(* Logix 5000 project; controller ACIM5010ConveyorHailee_Renkers vendor 1 type 14 code 77 rev 20.12; software revision 20.01 *)

TASK MainTask (continuous, watchdog 500 ms) : MainProgram

MODULES
   Controller : vendor 1 type 14 code 77 (CompactLogixL32EController 0, rev 20.12)
      LocalENB : 1769-L32E Ethernet Port (CompactLogixL32Ethernet 1, rev 20.11)
      Local : CompactBus (CompactVirtualAdapter 3, rev 20.11)
         Inputmod : 1769-IQ16 (Compact 1, rev 1.1, Input RPI 20 ms)
         OutputMod : 1769-OW16 (Compact 2, rev 1.1, Output RPI 20 ms)
END_MODULES

VAR_GLOBAL   (* controller tags *)
   Bin_Left_Red_Light : ALIAS FOR Local:2:O.Data.3;
   Bin_Right_Red_Light : ALIAS FOR Local:2:O.Data.4;
   CONVEYOR_AUX : ALIAS FOR Local:1:I.Data.12;
   CONVEYOR_MOTOR : ALIAS FOR Local:2:O.Data.2;
   FORWARD_AUX : ALIAS FOR Local:1:I.Data.10;
   FORWARD_MOTOR : ALIAS FOR Local:2:O.Data.0;
   GREEN_LIGHT : ALIAS FOR Local:2:O.Data.6;
   Limit_Switch_Left : ALIAS FOR Local:1:I.Data.13;
   Limit_Switch_Right : ALIAS FOR Local:1:I.Data.14;
   PHOTOEYE : ALIAS FOR Local:1:I.Data.15;
   REVERSE_AUX : ALIAS FOR Local:1:I.Data.11;
   REVERSE_MOTOR : ALIAS FOR Local:2:O.Data.1;
   START_PB : ALIAS FOR Local:1:I.Data.9;
   STOP_PB : ALIAS FOR Local:1:I.Data.8;
   YELLOW_LIGHT : ALIAS FOR Local:2:O.Data.5;
END_VAR

PROGRAM MainProgram   (* main routine MainRoutine *)
VAR
   counter : COUNTER := (PRE := 4);
   done : COUNTER := (PRE := 4);
   Latch : BOOL;
   Latch2 : BOOL;
   left : BOOL;
   left_bit_check : BOOL;
   left_latch : BOOL;
   lls_i : BOOL;
   OFF_DELAY : TIMER := (PRE := 1000);
   ON_DELAY : TIMER := (PRE := 1000);
   ONESHOTTIMER : BOOL;
   PI_Counter : COUNTER := (PRE := 8);
   pie_i : BOOL;
   PROCESS_COUNTER : COUNTER := (PRE := 4);
   right : BOOL;
   right_bit_check : BOOL;
   right_latch : BOOL;
   rls_i : BOOL;
   S0 : BOOL;
   S0_x : BOOL;
   S1 : BOOL;
   S1_x : BOOL;
   S2 : BOOL;
   S2_x : BOOL;
   S3 : BOOL;
   S3_x : BOOL;
   S4 : BOOL;
   S4_x : BOOL;
   S5 : BOOL;
   S5_x : BOOL;
   S6 : BOOL;
   S6_x : BOOL;
   start_i : BOOL;
   stop_i : BOOL;
END_VAR

ROUTINE MainRoutine   (* ladder *)
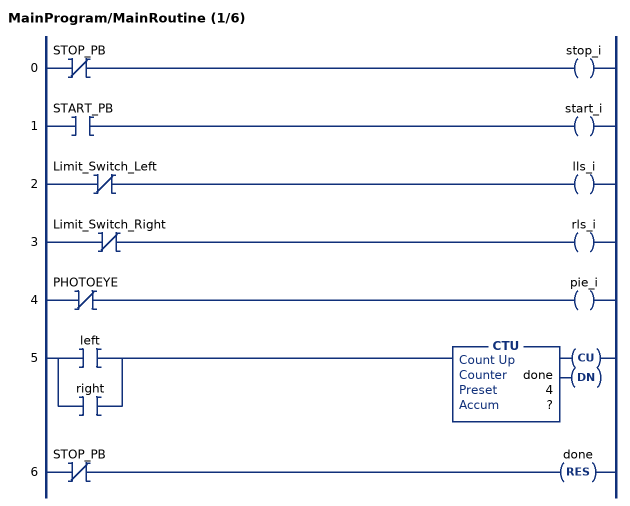
   0: XIO(STOP_PB)OTE(stop_i);
   1: XIC(START_PB)OTE(start_i);
   2: XIO(Limit_Switch_Left)OTE(lls_i);
   3: XIO(Limit_Switch_Right)OTE(rls_i);
   4: XIO(PHOTOEYE)OTE(pie_i);
   5: [XIC(left) ,XIC(right) ]CTU(done,?,?);
   6: XIO(STOP_PB)RES(done);
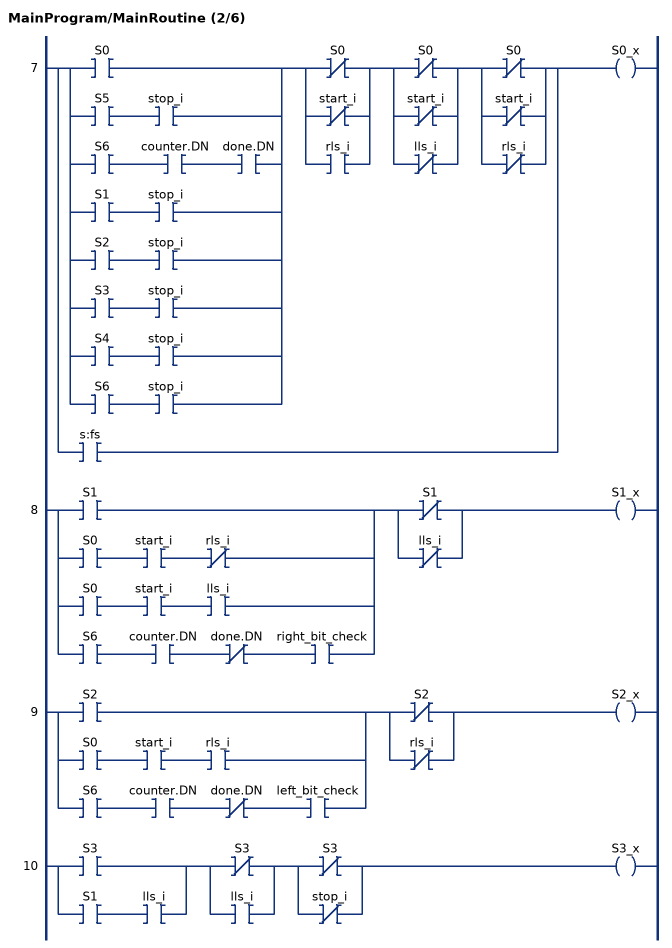
   7: [[XIC(S0) ,XIC(S5) XIC(stop_i) ,XIC(S6) XIC(counter.DN) XIC(done.DN) ,XIC(S1) XIC(stop_i) ,XIC(S2) XIC(stop_i) ,XIC(S3) XIC(stop_i) ,XIC(S4) XIC(stop_i) ,XIC(S6) XIC(stop_i) ] [XIO(S0) ,XIO(start_i) ,XIC(rls_i) ] [XIO(S0) ,XIO(start_i) ,XIO(lls_i) ] [XIO(S0) ,XIO(start_i) ,XIO(rls_i) ] ,XIC(s:fs) ]OTE(S0_x);
   8: [XIC(S1) ,[XIC(S0) XIC(start_i) XIO(rls_i) ,XIC(S0) XIC(start_i) XIC(lls_i) ] ,XIC(S6) XIC(counter.DN) XIO(done.DN) XIC(right_bit_check) ][XIO(S1) ,XIO(lls_i) ]OTE(S1_x);
   9: [XIC(S2) ,XIC(S0) XIC(start_i) XIC(rls_i) ,XIC(S6) XIC(counter.DN) XIO(done.DN) XIC(left_bit_check) ][XIO(S2) ,XIO(rls_i) ]OTE(S2_x);
   10: [XIC(S3) ,XIC(S1) XIC(lls_i) ][XIO(S3) ,XIC(lls_i) ][XIO(S3) ,XIO(stop_i) ]OTE(S3_x);
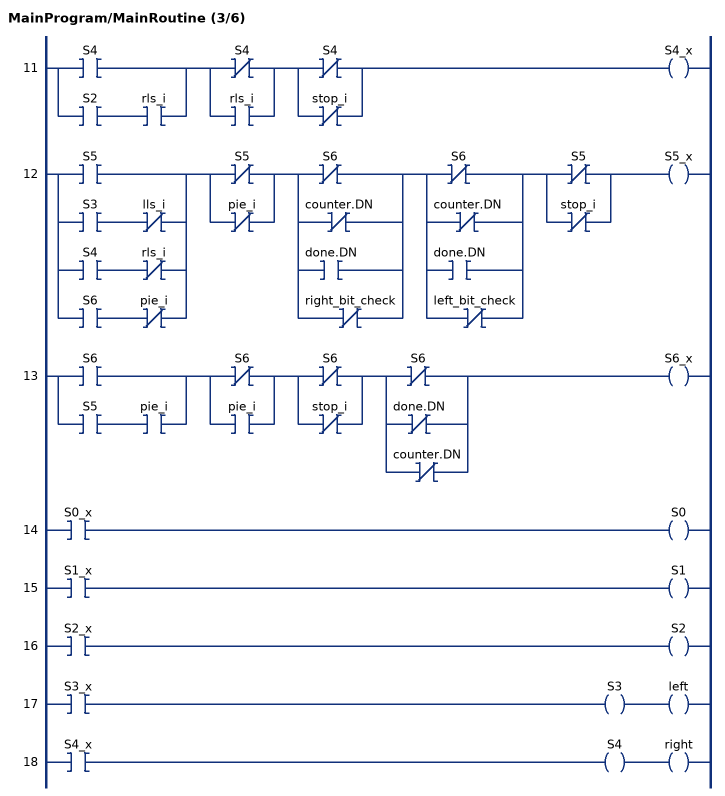
   11: [XIC(S4) ,XIC(S2) XIC(rls_i) ][XIO(S4) ,XIC(rls_i) ][XIO(S4) ,XIO(stop_i) ]OTE(S4_x);
   12: [XIC(S5) ,XIC(S3) XIO(lls_i) ,XIC(S4) XIO(rls_i) ,XIC(S6) XIO(pie_i) ][XIO(S5) ,XIO(pie_i) ][XIO(S6) ,XIO(counter.DN) ,XIC(done.DN) ,XIO(right_bit_check) ][XIO(S6) ,XIO(counter.DN) ,XIC(done.DN) ,XIO(left_bit_check) ][XIO(S5) ,XIO(stop_i) ]OTE(S5_x);
   13: [XIC(S6) ,XIC(S5) XIC(pie_i) ][XIO(S6) ,XIC(pie_i) ][XIO(S6) ,XIO(stop_i) ][XIO(S6) ,XIO(done.DN) ,XIO(counter.DN) ]OTE(S6_x);
   14: XIC(S0_x)OTE(S0);
   15: XIC(S1_x)OTE(S1);
   16: XIC(S2_x)OTE(S2);
   17: XIC(S3_x)OTE(S3)OTE(left);
   18: XIC(S4_x)OTE(S4)OTE(right);
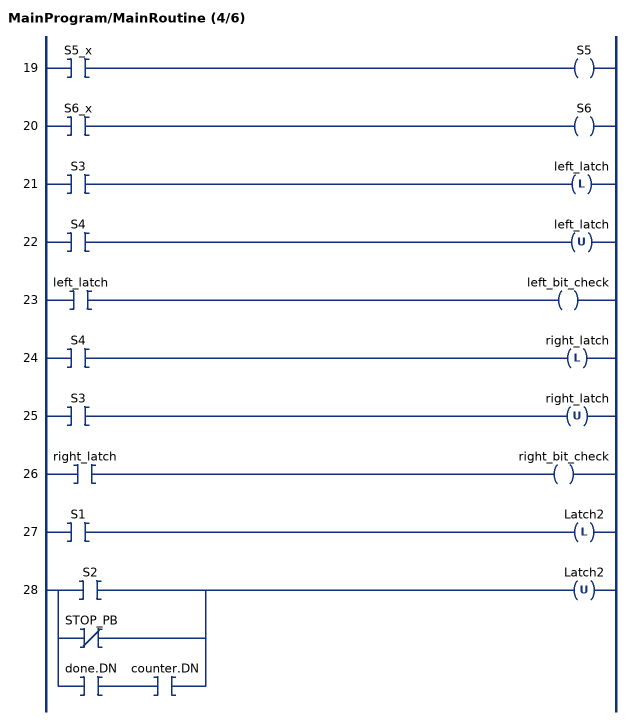
   19: XIC(S5_x)OTE(S5);
   20: XIC(S6_x)OTE(S6);
   21: XIC(S3)OTL(left_latch);
   22: XIC(S4)OTU(left_latch);
   23: XIC(left_latch)OTE(left_bit_check);
   24: XIC(S4)OTL(right_latch);
   25: XIC(S3)OTU(right_latch);
   26: XIC(right_latch)OTE(right_bit_check);
   27: XIC(S1)OTL(Latch2);
   28: [XIC(S2) ,XIO(STOP_PB) ,XIC(done.DN) XIC(counter.DN) ]OTU(Latch2);
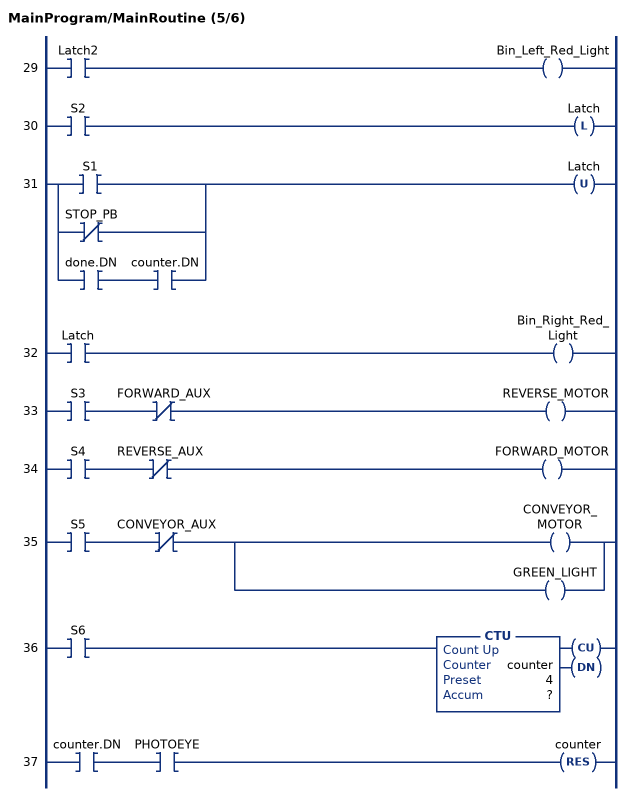
   29: XIC(Latch2)OTE(Bin_Left_Red_Light);
   30: XIC(S2)OTL(Latch);
   31: [XIC(S1) ,XIO(STOP_PB) ,XIC(done.DN) XIC(counter.DN) ]OTU(Latch);
   32: XIC(Latch)OTE(Bin_Right_Red_Light);
   33: XIC(S3)XIO(FORWARD_AUX)OTE(REVERSE_MOTOR);
   34: XIC(S4)XIO(REVERSE_AUX)OTE(FORWARD_MOTOR);
   35: XIC(S5)XIO(CONVEYOR_AUX)[OTE(CONVEYOR_MOTOR) ,OTE(GREEN_LIGHT) ];
   36: XIC(S6)CTU(counter,?,?);
   37: XIC(counter.DN)XIC(PHOTOEYE)RES(counter);
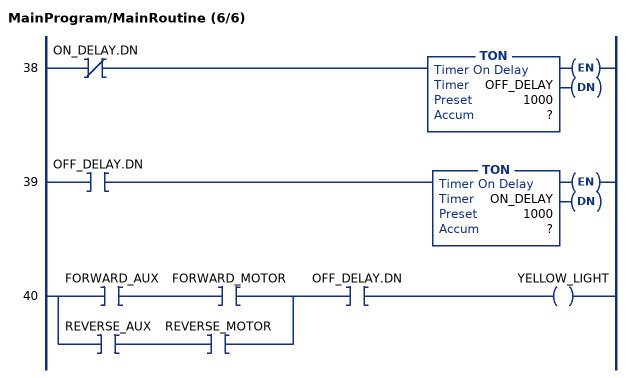
   38: XIO(ON_DELAY.DN)TON(OFF_DELAY,?,?);
   39: XIC(OFF_DELAY.DN)TON(ON_DELAY,?,?);
   40: [XIC(FORWARD_AUX) XIC(FORWARD_MOTOR) ,XIC(REVERSE_AUX) XIC(REVERSE_MOTOR) ]XIC(OFF_DELAY.DN)OTE(YELLOW_LIGHT);
END_ROUTINE
END_PROGRAM
